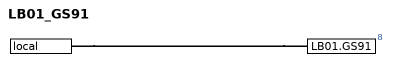
// note: 4 stored wires end on pins the file does not list and are not shown
local := LB01.GS91;
// Rotation heater guard trigged
AlarmAcknowledge01(Alarm := local.InputAlarm, InitPulse := SYS_InitPulse, AlarmAck := local.ACK); // _BE_AlarmAckRequired
local.AL01 := AlarmAcknowledge01.AlarmActive;
// Status HMI
IF true THEN _w1 := 0; END_IF
local.Symbol := _w1;
_w2 := local.AL01;
IF _w2 THEN _w3 := 2; END_IF
local.AL := _w2;
local.Symbol := _w3;
LB01.GS91 := local;
// al: input not connected

END_PROGRAM

// Device/AREA1/B001/LB01/Sequence/LB01_SequenceHeating
PROGRAM LB01_SequenceHeating
VAR
	nh_v: BOOL;
	seqMasterBreakpoint: LREAL;
	SequenceMaster: _BE_TwoSequenceMaster;
END_VAR

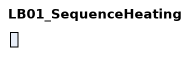
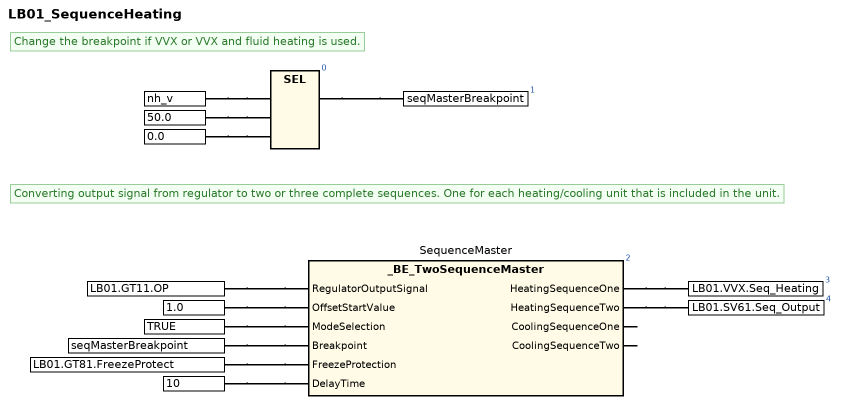
// Change the breakpoint if VVX or VVX and fluid heating is used.
seqMasterBreakpoint := SEL(nh_v, 50.0, 0.0);
// Converting output signal from regulator to two or three complete sequences. One for each heating/cooling unit that is included in the unit.
SequenceMaster(
    RegulatorOutputSignal := LB01.GT11.OP,
    OffsetStartValue := 1.0,
    ModeSelection := TRUE,
    Breakpoint := seqMasterBreakpoint,
    FreezeProtection := LB01.GT81.FreezeProtect,
    DelayTime := 10); // _BE_TwoSequenceMaster
LB01.VVX.Seq_Heating := SequenceMaster.HeatingSequenceOne;
LB01.SV61.Seq_Output := SequenceMaster.HeatingSequenceTwo;

END_PROGRAM

// Device/AREA1/B001/LB01/Sequence/LB01_SequenceCooling
PROGRAM LB01_SequenceCooling
VAR
	SequenceMaster: _BE_TwoSequenceMaster;
END_VAR
VAR // added by the converter: edge detectors and wires of the graphical bodies
    _w1 : BOOL;
    _w2, _w3 : ANY;
END_VAR

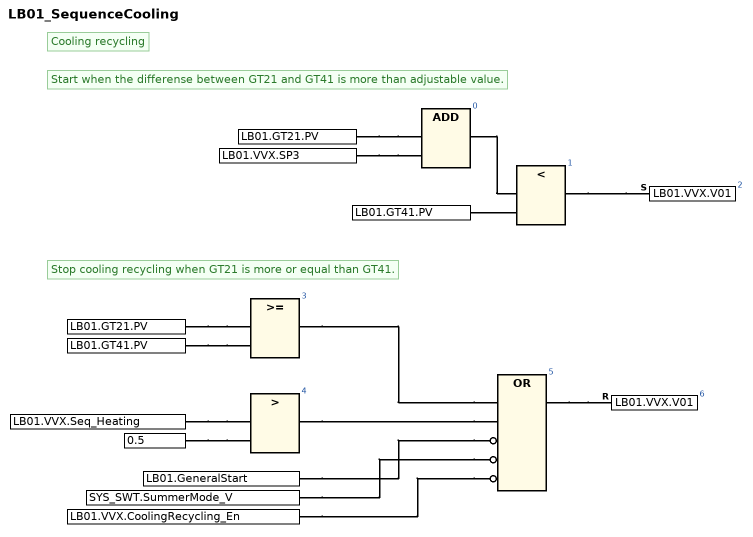
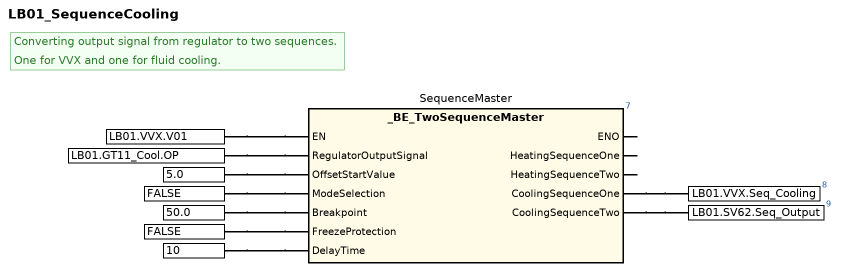
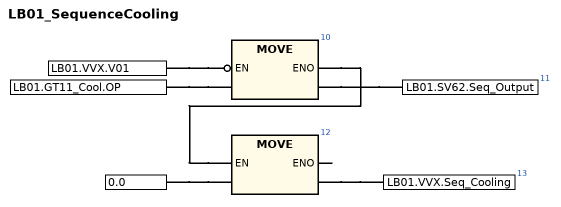
// Cooling recycling
// Start when the differense between GT21 and GT41 is more than adjustable value.
LB01.VVX.V01 S= LB01.GT21.PV + LB01.VVX.SP3 < LB01.GT41.PV;
// Stop cooling recycling when GT21 is more or equal than GT41.
LB01.VVX.V01 R= LB01.GT21.PV >= LB01.GT41.PV OR LB01.VVX.Seq_Heating > 0.5 OR NOT LB01.GeneralStart OR NOT SYS_SWT.SummerMode_V OR NOT LB01.VVX.CoolingRecycling_En;
// Converting output signal from regulator to two sequences.
// One for VVX and one for fluid cooling.
IF LB01.VVX.V01 THEN
    SequenceMaster(
        RegulatorOutputSignal := LB01.GT11_Cool.OP,
        OffsetStartValue := 5.0,
        ModeSelection := FALSE,
        Breakpoint := 50.0,
        FreezeProtection := FALSE,
        DelayTime := 10); // _BE_TwoSequenceMaster
END_IF
LB01.VVX.Seq_Cooling := SequenceMaster.CoolingSequenceOne;
LB01.SV62.Seq_Output := SequenceMaster.CoolingSequenceTwo;
_w1 := NOT LB01.VVX.V01;
IF _w1 THEN _w2 := LB01.GT11_Cool.OP; END_IF
LB01.SV62.Seq_Output := _w2;
IF _w1 THEN _w3 := 0.0; END_IF
LB01.VVX.Seq_Cooling := _w3;

END_PROGRAM

// Device/AREA1/B001/LB01/Sensor/Temperature/GT12/LB01_GT12
PROGRAM LB01_GT12
VAR
	local:strSensor1;
	gt_Min: TON;
	gt_Max: TON;
	ackFault: BOOL;
	ackLal: BOOL;
	ackHal: BOOL;
	AlarmAcknowledge01: _BE_AlarmAckRemote;
	AlarmAcknowledge02: _BE_AlarmAckRemote;
	AlarmAcknowledge03: _BE_AlarmAckRemote;
END_VAR
VAR // added by the converter: edge detectors and wires of the graphical bodies
    _w1, _w3, _w4 : ANY;
    _w2 : BOOL;
END_VAR

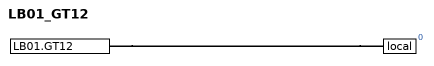
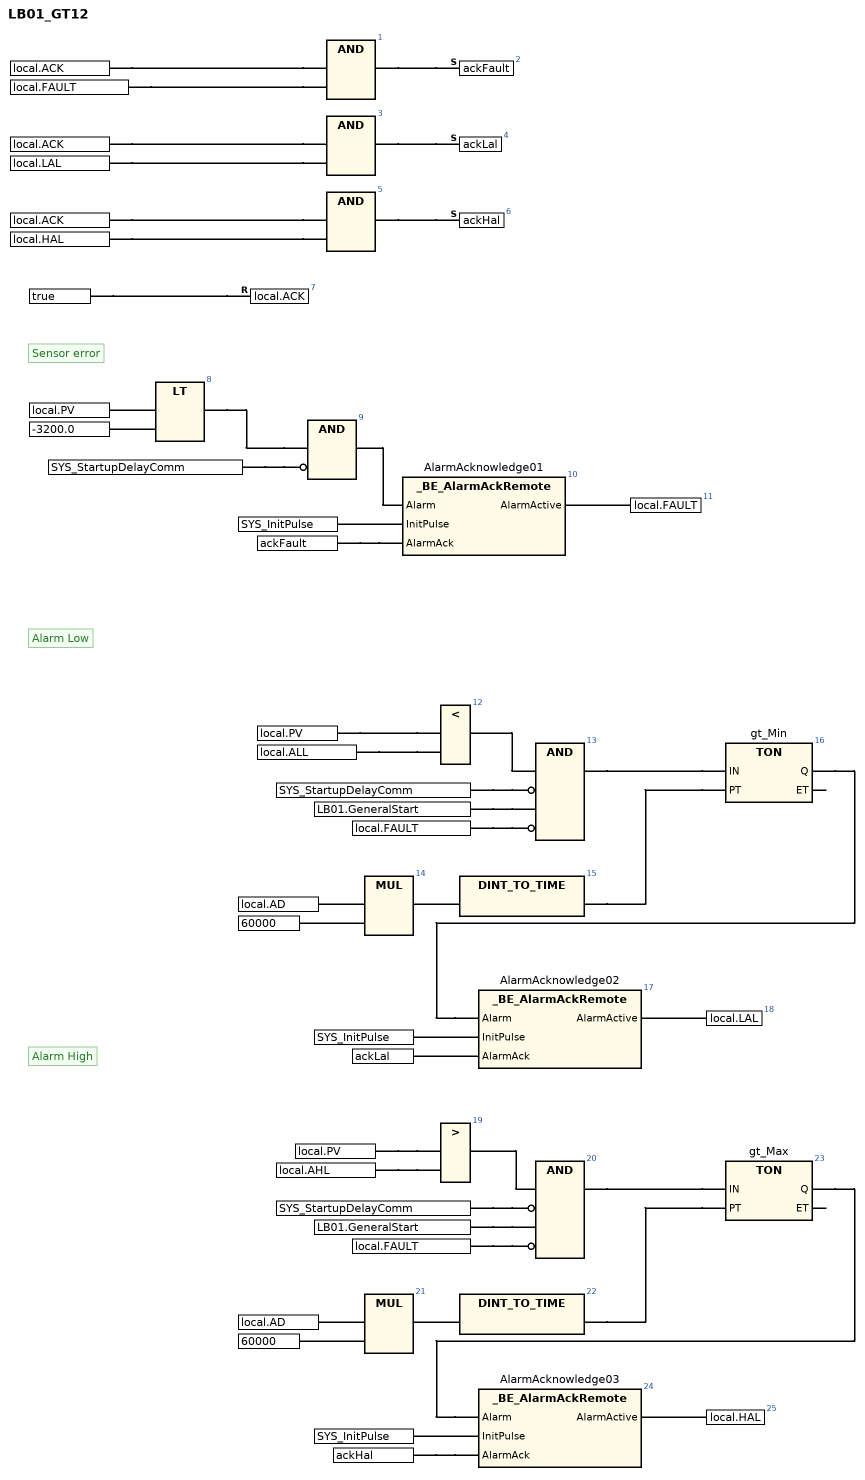
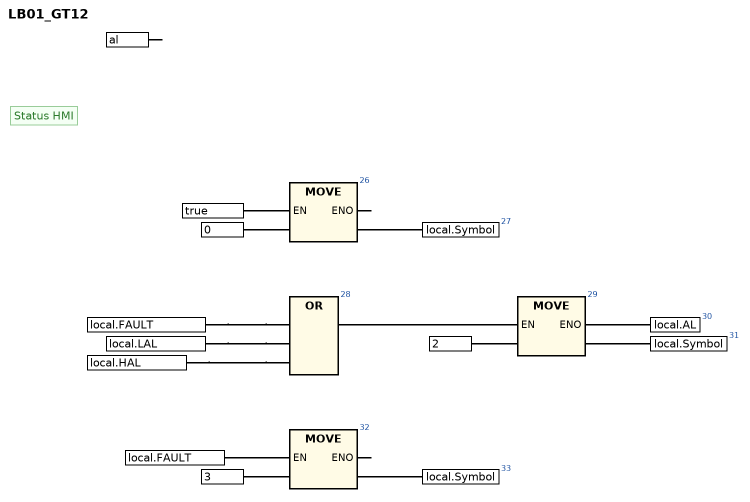
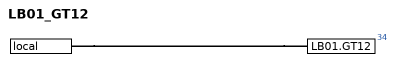
// note: 4 stored wires end on pins the file does not list and are not shown
local := LB01.GT12;
ackFault S= local.ACK AND local.FAULT;
ackLal S= local.ACK AND local.LAL;
ackHal S= local.ACK AND local.HAL;
local.ACK R= true;
// Sensor error
AlarmAcknowledge01(
    Alarm := local.PV < -3200.0 AND NOT SYS_StartupDelayComm,
    InitPulse := SYS_InitPulse,
    AlarmAck := ackFault); // _BE_AlarmAckRemote
local.FAULT := AlarmAcknowledge01.AlarmActive;
// Alarm Low
gt_Min(IN := local.PV < local.ALL AND NOT SYS_StartupDelayComm AND LB01.GeneralStart AND NOT local.FAULT, PT := DINT_TO_TIME(local.AD * 60000)); // TON
AlarmAcknowledge02(Alarm := gt_Min.Q, InitPulse := SYS_InitPulse, AlarmAck := ackLal); // _BE_AlarmAckRemote
local.LAL := AlarmAcknowledge02.AlarmActive;
// Alarm High
gt_Max(IN := local.PV > local.AHL AND NOT SYS_StartupDelayComm AND LB01.GeneralStart AND NOT local.FAULT, PT := DINT_TO_TIME(local.AD * 60000)); // TON
AlarmAcknowledge03(Alarm := gt_Max.Q, InitPulse := SYS_InitPulse, AlarmAck := ackHal); // _BE_AlarmAckRemote
local.HAL := AlarmAcknowledge03.AlarmActive;
// Status HMI
IF true THEN _w1 := 0; END_IF
local.Symbol := _w1;
_w2 := local.FAULT OR local.LAL OR local.HAL;
IF _w2 THEN _w3 := 2; END_IF
local.AL := _w2;
local.Symbol := _w3;
IF local.FAULT THEN _w4 := 3; END_IF
local.Symbol := _w4;
LB01.GT12 := local;
// al: input not connected

END_PROGRAM

// Device/AREA1/B001/LB01/Sensor/Temperature/GT13/LB01_GT13
PROGRAM LB01_GT13
VAR
	local:strSensor1;
	gt_Min: TON;
	gt_Max: TON;
	ackFault: BOOL;
	ackLal: BOOL;
	ackHal: BOOL;
	AlarmAcknowledge01: _BE_AlarmAckRemote;
	AlarmAcknowledge02: _BE_AlarmAckRemote;
	AlarmAcknowledge03: _BE_AlarmAckRemote;
END_VAR
VAR // added by the converter: edge detectors and wires of the graphical bodies
    _w1, _w3, _w4 : ANY;
    _w2 : BOOL;
END_VAR

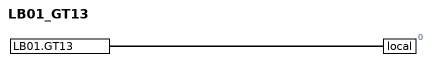
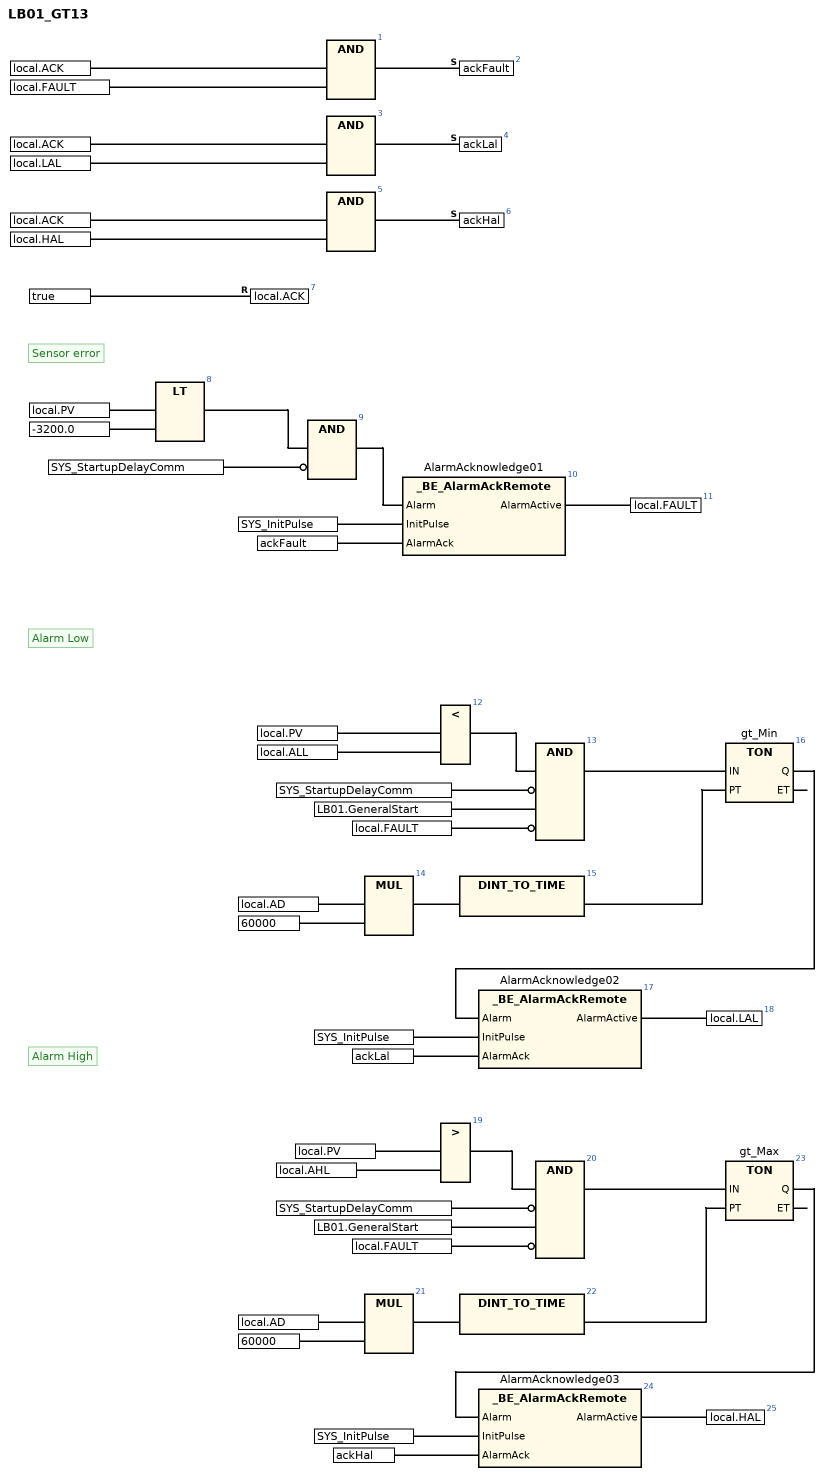
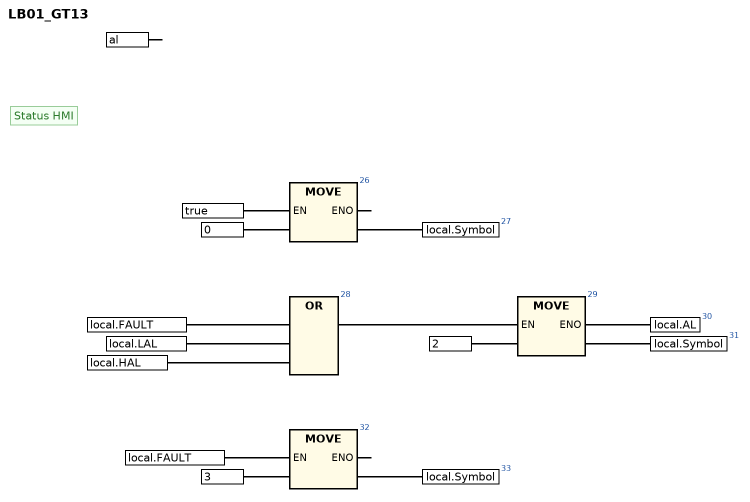
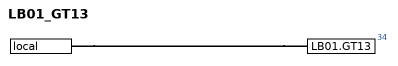
// note: 4 stored wires end on pins the file does not list and are not shown
local := LB01.GT13;
ackFault S= local.ACK AND local.FAULT;
ackLal S= local.ACK AND local.LAL;
ackHal S= local.ACK AND local.HAL;
local.ACK R= true;
// Sensor error
AlarmAcknowledge01(
    Alarm := local.PV < -3200.0 AND NOT SYS_StartupDelayComm,
    InitPulse := SYS_InitPulse,
    AlarmAck := ackFault); // _BE_AlarmAckRemote
local.FAULT := AlarmAcknowledge01.AlarmActive;
// Alarm Low
gt_Min(IN := local.PV < local.ALL AND NOT SYS_StartupDelayComm AND LB01.GeneralStart AND NOT local.FAULT, PT := DINT_TO_TIME(local.AD * 60000)); // TON
AlarmAcknowledge02(Alarm := gt_Min.Q, InitPulse := SYS_InitPulse, AlarmAck := ackLal); // _BE_AlarmAckRemote
local.LAL := AlarmAcknowledge02.AlarmActive;
// Alarm High
gt_Max(IN := local.PV > local.AHL AND NOT SYS_StartupDelayComm AND LB01.GeneralStart AND NOT local.FAULT, PT := DINT_TO_TIME(local.AD * 60000)); // TON
AlarmAcknowledge03(Alarm := gt_Max.Q, InitPulse := SYS_InitPulse, AlarmAck := ackHal); // _BE_AlarmAckRemote
local.HAL := AlarmAcknowledge03.AlarmActive;
// Status HMI
IF true THEN _w1 := 0; END_IF
local.Symbol := _w1;
_w2 := local.FAULT OR local.LAL OR local.HAL;
IF _w2 THEN _w3 := 2; END_IF
local.AL := _w2;
local.Symbol := _w3;
IF local.FAULT THEN _w4 := 3; END_IF
local.Symbol := _w4;
LB01.GT13 := local;
// al: input not connected

END_PROGRAM

// Device/AREA1/B001/LB01/Sensor/Temperature/GT22/LB01_GT22
PROGRAM LB01_GT22
VAR
	local:strSensor1;
	gt_Min: TON;
	gt_Max: TON;
	ackFault: BOOL;
	ackLal: BOOL;
	ackHal: BOOL;
	AlarmAcknowledge01: _BE_AlarmAckRemote;
	AlarmAcknowledge02: _BE_AlarmAckRemote;
	AlarmAcknowledge03: _BE_AlarmAckRemote;
END_VAR
VAR // added by the converter: edge detectors and wires of the graphical bodies
    _w1, _w3, _w4 : ANY;
    _w2 : BOOL;
END_VAR

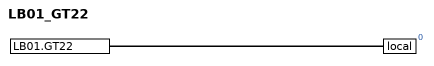
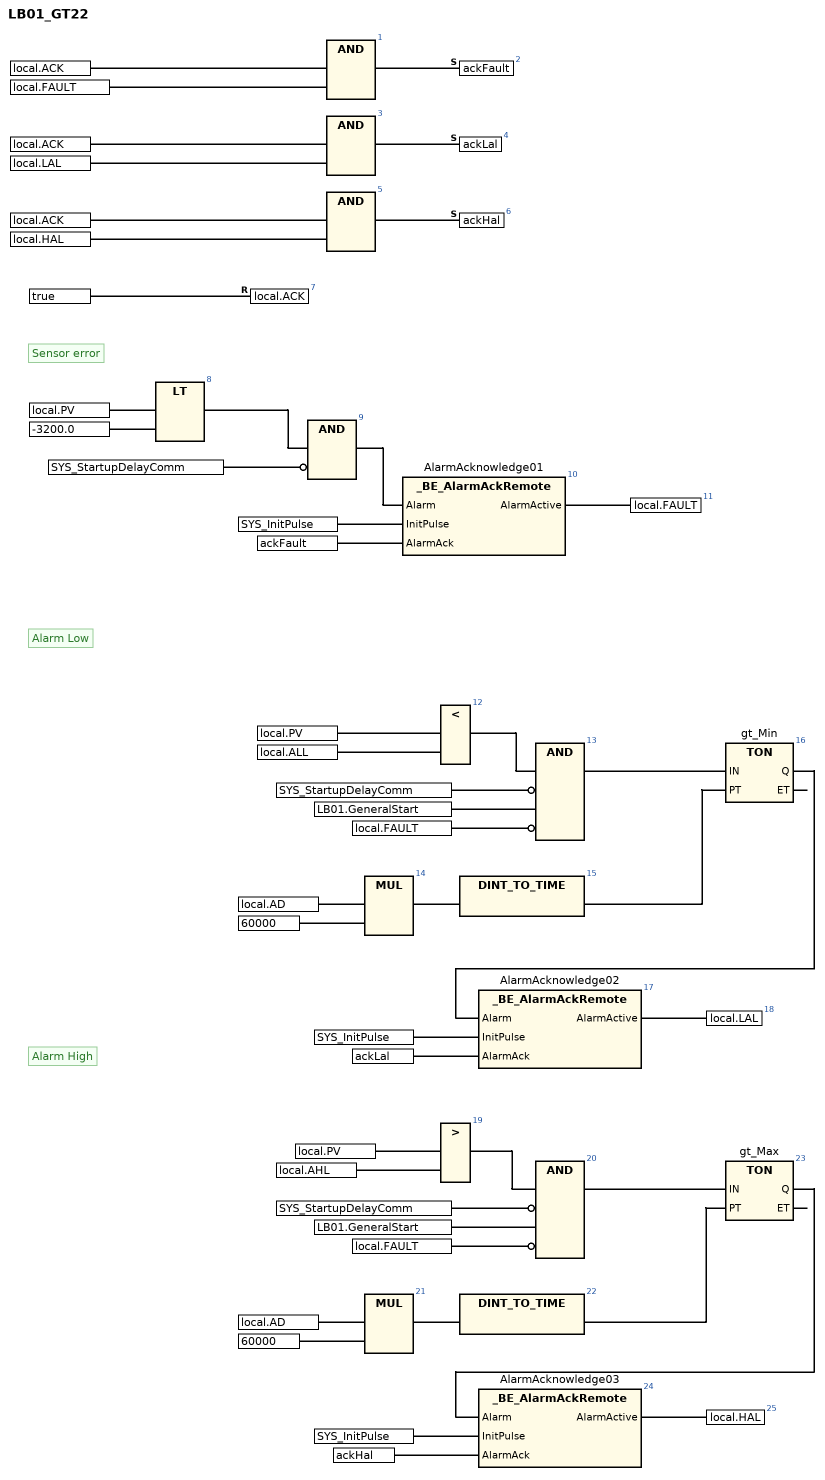
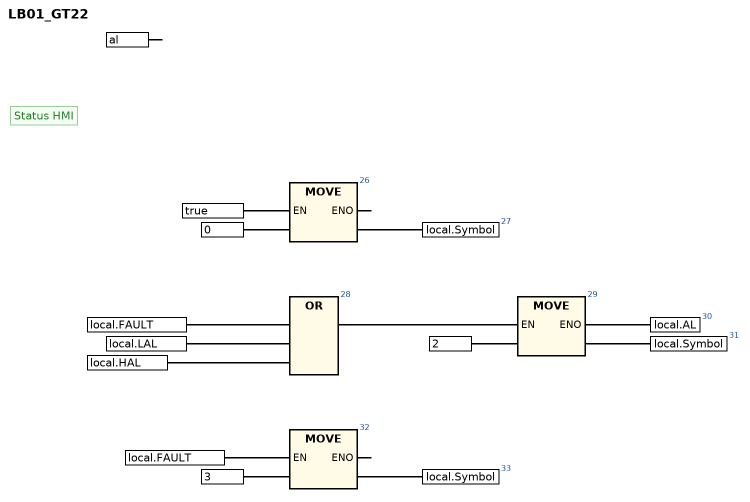
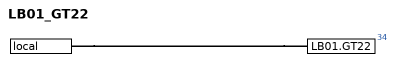
// note: 4 stored wires end on pins the file does not list and are not shown
local := LB01.GT22;
ackFault S= local.ACK AND local.FAULT;
ackLal S= local.ACK AND local.LAL;
ackHal S= local.ACK AND local.HAL;
local.ACK R= true;
// Sensor error
AlarmAcknowledge01(
    Alarm := local.PV < -3200.0 AND NOT SYS_StartupDelayComm,
    InitPulse := SYS_InitPulse,
    AlarmAck := ackFault); // _BE_AlarmAckRemote
local.FAULT := AlarmAcknowledge01.AlarmActive;
// Alarm Low
gt_Min(IN := local.PV < local.ALL AND NOT SYS_StartupDelayComm AND LB01.GeneralStart AND NOT local.FAULT, PT := DINT_TO_TIME(local.AD * 60000)); // TON
AlarmAcknowledge02(Alarm := gt_Min.Q, InitPulse := SYS_InitPulse, AlarmAck := ackLal); // _BE_AlarmAckRemote
local.LAL := AlarmAcknowledge02.AlarmActive;
// Alarm High
gt_Max(IN := local.PV > local.AHL AND NOT SYS_StartupDelayComm AND LB01.GeneralStart AND NOT local.FAULT, PT := DINT_TO_TIME(local.AD * 60000)); // TON
AlarmAcknowledge03(Alarm := gt_Max.Q, InitPulse := SYS_InitPulse, AlarmAck := ackHal); // _BE_AlarmAckRemote
local.HAL := AlarmAcknowledge03.AlarmActive;
// Status HMI
IF true THEN _w1 := 0; END_IF
local.Symbol := _w1;
_w2 := local.FAULT OR local.LAL OR local.HAL;
IF _w2 THEN _w3 := 2; END_IF
local.AL := _w2;
local.Symbol := _w3;
IF local.FAULT THEN _w4 := 3; END_IF
local.Symbol := _w4;
LB01.GT22 := local;
// al: input not connected

END_PROGRAM

// Device/AREA1/B001/LB01/Function/LB01_Function_Dewpoint
PROGRAM LB01_Function_Dewpoint
VAR
	FbDewPoint: _BE_DewTemperaturePoint;
END_VAR

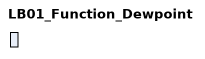
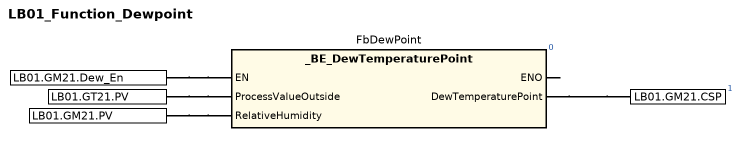
IF LB01.GM21.Dew_En THEN
    FbDewPoint(ProcessValueOutside := LB01.GT21.PV, RelativeHumidity := LB01.GM21.PV); // _BE_DewTemperaturePoint
END_IF
LB01.GM21.CSP := FbDewPoint.DewTemperaturePoint;

END_PROGRAM

// Device/AREA1/B001/LB01/Function/LB01_Function_EfficiencyExtractAir
PROGRAM LB01_Function_EfficiencyExtractAir
VAR
	FbEfficiency: _BE_RecoveryEfficiencyExtractAir;
	gt_Min: TON;
	AlarmAcknowledge01: _BE_AlarmAckRemote;
END_VAR
VAR // added by the converter: edge detectors and wires of the graphical bodies
    _w1 : ANY;
END_VAR

